% RSLogix 500 project P6A_HOURMETER.RSS, saved by version 8.30.00.16 %
PROJECT "P6"    % processor: Bul.1763 MicroLogix 1100 Series B %

PROGRAM FILES
  LAD 2   9 rungs

DATA FILES
  O0 OUTPUT  4 elements
  I1 INPUT  6 elements
  S2 STATUS  66 elements
  B3 BINARY  1 elements
  T4 TIMER  1 elements
  C5 COUNTER  5 elements
  R6 CONTROL  1 elements
  N7 INTEGER  15 elements
  F8 FLOAT  1 elements

LADDER 2
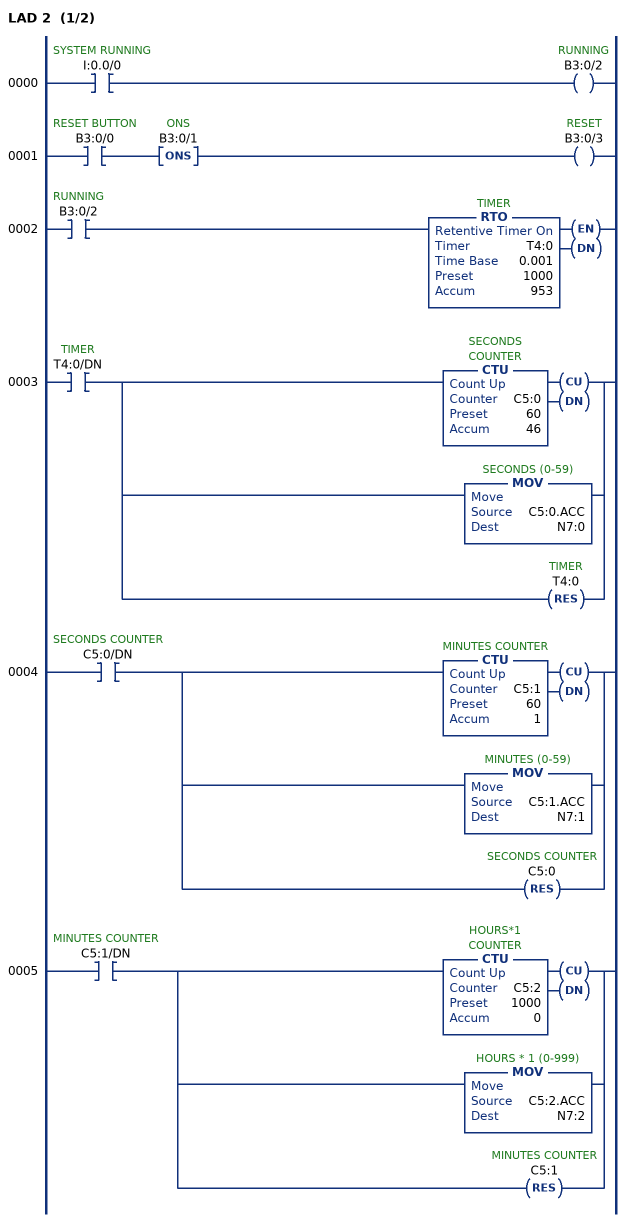
% Rung: 0 %
SOR XIC I:0.0/0 OTE B3:0/2 EOR
%   I:0.0/0  "SYSTEM RUNNING" %
%   B3:0/2  "RUNNING" %
% Rung: 1 %
SOR XIC B3:0/0 ONS B3:0/1 OTE B3:0/3 EOR
%   B3:0/0  "RESET BUTTON" %
%   B3:0/1  "ONS" %
%   B3:0/3  "RESET" %
% Rung: 2 %
SOR XIC B3:0/2 RTO T4:0 0.001 1000 953 EOR
%   B3:0/2  "RUNNING" %
%   T4:0  "TIMER" %
% Rung: 3 %
SOR XIC T4:0/DN BST CTU C5:0 60 46 NXB MOV C5:0.ACC N7:0 NXB RES T4:0 BND EOR
%   T4:0  "TIMER" %
%   C5:0  "SECONDS COUNTER" %
%   N7:0  "SECONDS (0-59)" %
% Rung: 4 %
SOR XIC C5:0/DN BST CTU C5:1 60 1 NXB MOV C5:1.ACC N7:1 NXB RES C5:0 BND EOR
%   C5:0  "SECONDS COUNTER" %
%   C5:1  "MINUTES COUNTER" %
%   N7:1  "MINUTES (0-59)" %
% Rung: 5 %
SOR XIC C5:1/DN BST CTU C5:2 1000 0 NXB MOV C5:2.ACC N7:2 NXB RES C5:1 BND EOR
%   C5:1  "MINUTES COUNTER" %
%   C5:2  "HOURS*1 COUNTER" %
%   N7:2  "HOURS * 1 (0-999)" %

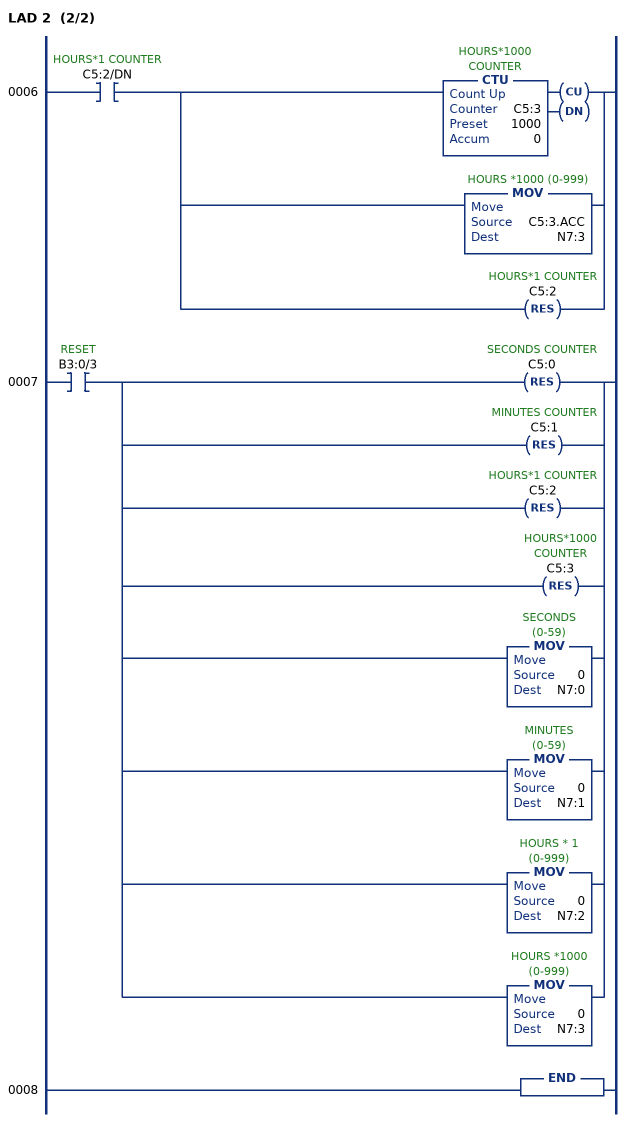
% Rung: 6 %
SOR XIC C5:2/DN BST CTU C5:3 1000 0 NXB MOV C5:3.ACC N7:3 NXB RES C5:2 BND EOR
%   C5:2  "HOURS*1 COUNTER" %
%   C5:3  "HOURS*1000 COUNTER" %
%   N7:3  "HOURS *1000 (0-999)" %
% Rung: 7 %
SOR XIC B3:0/3 BST RES C5:0 NXB RES C5:1 NXB RES C5:2 NXB RES C5:3 NXB MOV 0 N7:0 NXB MOV 0 N7:1 NXB MOV 0 N7:2 NXB MOV 0 N7:3 BND EOR
%   B3:0/3  "RESET" %
%   C5:0  "SECONDS COUNTER" %
%   C5:1  "MINUTES COUNTER" %
%   C5:2  "HOURS*1 COUNTER" %
%   C5:3  "HOURS*1000 COUNTER" %
%   N7:0  "SECONDS (0-59)" %
%   N7:1  "MINUTES (0-59)" %
%   N7:2  "HOURS * 1 (0-999)" %
%   N7:3  "HOURS *1000 (0-999)" %
% Rung: 8 %
SOR END EOR

DATA TABLE (non-zero values as saved)
DATA B3
% B3:0 % 0X0004
DATA T4
% .PRE .ACC %
% T4:0 % 1000 953
DATA C5
% .PRE .ACC %
% C5:0 % 60 46
% C5:1 % 60 1
% C5:2 % 1000 0
% C5:3 % 1000 0
DATA N7
% N7:0 % 46 1 0 0 0 0 0 0 0 0
